KUKA KRL data list: RotinaATIVOS.dat

&ACCESS RV
DEFDAT RotinaATIVOS

ENDDAT
